FUNCTION_BLOCK FB_TM1K4
(*
    Adapted from FB_ATM to:
    - Change stTarget1..stTarget5 to stTarget1a, stTarget1b, stTarget2b, stTarget3a, stTarget3b, stTarget4, stTarget5 to the inputs
    - Change the arrStates.array pragma from 1..6 to 1..8 (out and 7 in states, up from 5)
    - Swap out FB_ATM_States for FB_TM1K4_States
*)
VAR_IN_OUT
    // Y motor (state select).
    stYStage: ST_MotionStage;
    // X motor (align target to beam).
    stXStage: ST_MotionStage;
    // The fast fault output to fault to.
    fbFFHWO: FB_HardwareFFOutput;
    // The arbiter to request beam conditions from.
    fbArbiter: FB_Arbiter;
END_VAR
VAR_INPUT
    stOut: ST_PositionState;
    stTarget1a: ST_PositionState;
    stTarget1b: ST_PositionState;
    stTarget2a: ST_PositionState;
    stTarget2b: ST_PositionState;
    stTarget3a: ST_PositionState;
    stTarget3b: ST_PositionState;
    stTarget4: ST_PositionState;    // target 4 is Yag
    stTarget5: ST_PositionState;    //target 5 is Diode
    // Set this to a non-unknown value to request a new move.
    {attribute 'pytmc' := '
        pv: MMS:STATE:SET
        io: io
    '}
    eEnumSet: ENUM_TM1K4_States;
    // Set this to TRUE to enable input state moves, or FALSE to disable them.
    bEnableMotion: BOOL;
    // Set this to TRUE to enable beam parameter checks, or FALSE to disable them.
    bEnableBeamParams: BOOL;
    // Set this to TRUE to enable position limit checks, or FALSE to disable them.
    bEnablePositionLimits: BOOL;
    // The name of the device for use in the PMPS DB lookup and diagnostic screens.
    sDeviceName: STRING;
    // The name of the transition state in the PMPS database.
    sTransitionKey: STRING;
    // Set this to TRUE to re-read the loaded database immediately (useful for debug).
    bReadDBNow: BOOL;
END_VAR
VAR_OUTPUT
    // The current position state as an enum.
    {attribute 'pytmc' := '
        pv: MMS:STATE:GET
        io: i
    '}
    eEnumGet: ENUM_TM1K4_States;
    // The PMPS database lookup associated with the current position state.
    stDbStateParams: ST_DbStateParams;
END_VAR
VAR
    bInit: BOOL;

    fbYStage: FB_MotionStage;
    fbXStage: FB_MotionStage;

    fbStateDefaults: FB_PositionState_Defaults;

    {attribute 'pytmc' := '
        pv: MMS
        astPositionState.array: 1..8
    '}
    fbStates: FB_PositionStatePMPS1D;
    astPositionState: ARRAY[1..GeneralConstants.MAX_STATES] OF ST_PositionState;
    fbArrCheckWrite: FB_CheckPositionStateWrite;

    {attribute 'pytmc' := 'pv: STC:01'}
    fbTempSensor1: FB_CC_TempSensor;

    {attribute 'pytmc' :='pv: FWM'}
    fbFlowMeter: FB_AnalogInput := (iTermBits:=15, fTermMax:=60, fTermMin:=0);
END_VAR
VAR CONSTANT
    // State defaults if not provided
    fDelta: LREAL := 2;
    fAccel: LREAL := 200;
    fOutDecel: LREAL := 25;
END_VAR

IF NOT bInit THEN
    bInit := TRUE;

    stYStage.nEnableMode := ENUM_StageEnableMode.DURING_MOTION;
    stXStage.nEnableMode := ENUM_StageEnableMode.DURING_MOTION;

    // Partial backcompat, this used to set fVelocity too but this should be set per install
    fbStateDefaults(stPositionState:=stOut, sNameDefault:='OUT', fDeltaDefault:=fDelta, fAccelDefault:=fAccel, fDecelDefault:=fOutDecel);
    fbStateDefaults(stPositionState:=stTarget1a, sNameDefault:='TARGET1a', fDeltaDefault:=fDelta, fAccelDefault:=fAccel, fDecelDefault:=fAccel);
    fbStateDefaults(stPositionState:=stTarget1b, sNameDefault:='TARGET1b', fDeltaDefault:=fDelta, fAccelDefault:=fAccel, fDecelDefault:=fAccel);
    fbStateDefaults(stPositionState:=stTarget2a, sNameDefault:='TARGET2a', fDeltaDefault:=fDelta, fAccelDefault:=fAccel, fDecelDefault:=fAccel);
    fbStateDefaults(stPositionState:=stTarget2b, sNameDefault:='TARGET2b', fDeltaDefault:=fDelta, fAccelDefault:=fAccel, fDecelDefault:=fAccel);
    fbStateDefaults(stPositionState:=stTarget3a, sNameDefault:='TARGET3a', fDeltaDefault:=fDelta, fAccelDefault:=fAccel, fDecelDefault:=fAccel);
    fbStateDefaults(stPositionState:=stTarget3b, sNameDefault:='TARGET3b', fDeltaDefault:=fDelta, fAccelDefault:=fAccel, fDecelDefault:=fAccel);
    fbStateDefaults(stPositionState:=stTarget4, sNameDefault:='YAG', fDeltaDefault:=fDelta, fAccelDefault:=fAccel, fDecelDefault:=fAccel);
    fbStateDefaults(stPositionState:=stTarget5, sNameDefault:='DIODE', fDeltaDefault:=fDelta, fAccelDefault:=fAccel, fDecelDefault:=fAccel);
END_IF

stYStage.bHardwareEnable := TRUE;
stYStage.bPowerSelf := FALSE;

stXStage.bLimitForwardEnable := TRUE;
stXStage.bLimitBackwardEnable := TRUE;
stXStage.bHardwareEnable := TRUE;
stXStage.bPowerSelf := TRUE;

fbYStage(stMotionStage:=stYStage);
fbXStage(stMotionStage:=stXStage);

// We need to update from PLC or from EPICS, but not both
fbArrCheckWrite(
    astPositionState:=astPositionState,
    bCheck:=TRUE,
    bSave:=FALSE,
);
IF NOT fbArrCheckWrite.bHadWrite THEN
    astPositionState[ENUM_TM1K4_States.OUT] := stOut;
    astPositionState[ENUM_TM1K4_States.TARGET1a] := stTarget1a;
    astPositionState[ENUM_TM1K4_States.TARGET1b] := stTarget1b;
    astPositionState[ENUM_TM1K4_States.TARGET2a] := stTarget2a;
    astPositionState[ENUM_TM1K4_States.TARGET2b] := stTarget2b;
    astPositionState[ENUM_TM1K4_States.TARGET3a] := stTarget3a;
    astPositionState[ENUM_TM1K4_States.TARGET3b] := stTarget3b;
    astPositionState[ENUM_TM1K4_States.YAG] := stTarget4;
    astPositionState[ENUM_TM1K4_States.DIODE] := stTarget5;
END_IF

fbStates(
    stMotionStage:=stYStage,
    astPositionState:=astPositionState,
    eEnumSet:=eEnumSet,
    eEnumGet:=eEnumGet,
    fbFFHWO:=fbFFHWO,
    fbArbiter:=fbArbiter,
    bEnableMotion:=bEnableMotion,
    bEnableBeamParams:=bEnableBeamParams,
    bEnablePositionLimits:=bEnablePositionLimits,
    sDeviceName:=sDeviceName,
    sTransitionKey:=sTransitionKey,
    bReadDBNow:=bReadDBNow,
    stDbStateParams=>stDbStateParams,
);

fbArrCheckWrite(
    astPositionState:=astPositionState,
    bCheck:=FALSE,
    bSave:=TRUE,
);

stOut := astPositionState[ENUM_TM1K4_States.OUT];
stTarget1a := astPositionState[ENUM_TM1K4_States.TARGET1a];
stTarget1b := astPositionState[ENUM_TM1K4_States.TARGET1b];
stTarget2a := astPositionState[ENUM_TM1K4_States.TARGET2a];
stTarget2b := astPositionState[ENUM_TM1K4_States.TARGET2b];
stTarget3a := astPositionState[ENUM_TM1K4_States.TARGET3a];
stTarget3b := astPositionState[ENUM_TM1K4_States.TARGET3b];
stTarget4 := astPositionState[ENUM_TM1K4_States.YAG];
stTarget5 := astPositionState[ENUM_TM1K4_States.DIODE];

fbTempSensor1(
    fFaultThreshold:=fbStates.stDbStateParams.stReactiveParams.nTempSP,
    bVeto:=eEnumGet = ENUM_TM1K4_States.OUT,
    sDevName:=sDeviceName,
    io_fbFFHWO:=fbFFHWO,
);
fbFlowMeter();

END_FUNCTION_BLOCK

(* stored: Version 1.1.0.1, ProductVersion 3.1.4024.12
   POU FB_TM1K4: Id {cc4ef3a5-22a4-4947-b9a9-d14630638b00}, SpecialFunc None *)
